FUNCTION_BLOCK MOD_ActivityCount (* Number of running skills from the +1/-1 activity channel *)
  (* Standard: 61499-2 *)
  (* Version 0.1, 2026-09-28, Project contributors, AAU Smart Production Lab *)
  PACKAGE modlib;
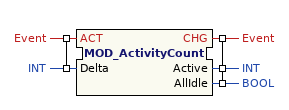
  EVENT_INPUT
    ACT WITH Delta;
  END_EVENT
  EVENT_OUTPUT
    CHG WITH Active, AllIdle;
  END_EVENT
  VAR_INPUT
    Delta : INT;
  END_VAR
  VAR_OUTPUT
    Active : INT;
    AllIdle : BOOL := TRUE;
  END_VAR
  EC_STATES
    ACT : ACT -> CHG;
  END_STATES
  ALGORITHM ACT IN ST:
Active := Active + Delta;
IF Active < 0 THEN
  Active := 0;
END_IF;
AllIdle := Active = 0;
  END_ALGORITHM
END_FUNCTION_BLOCK
